(* CoDeSys 2.3.9.50 project: 4A.pr6 *)
(* Libraries: STANDARD.LB6 5.6.98 12:03:02 *)

(* POU MAIN, LD *)
PROGRAM MAIN
VAR
	A AT %IX0.0: BOOL;
	C1: CTU;
	LightA AT %QX0.0: BOOL;
	C2: CTU;
	LightB AT %QX0.1: BOOL;
	Reset AT %IX0.3: BOOL;
END_VAR
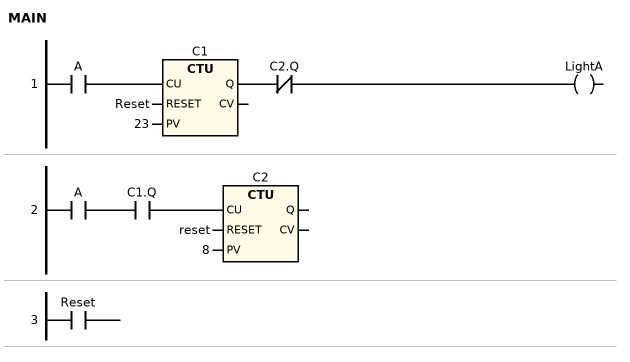
_LD_ (* Ladder Diagram *)
NETWORK 1
	[A] - C1:CTU(CU: *, RESET: Reset, PV: 23) - [/C2.Q] --- (LightA)
NETWORK 2
	[A] - [C1.Q] - C2:CTU(CU: *, RESET: reset, PV: 8)
NETWORK 3
	[Reset]
_END_LD_
(* the same logic as Structured Text *)
(* Network 1 *)
C1(CU := A, RESET := Reset, PV := 23);
LightA := C1.Q AND NOT C2.Q;
(* Network 2 *)
C2(CU := A AND C1.Q, RESET := reset, PV := 8);
(* Network 3 *)
END_PROGRAM
